{attribute 'qualified_only'}
VAR_GLOBAL
	
	// Termo-resistances outputs
	O_TermL:BOOL;
	O_TermU:BOOL;
END_VAR

(* stored: Version 1.1.0.1, ProductVersion 3.1.4024.9
   GVL IO: Id {f19c6e7d-dfbd-4478-b507-c13927482bf7} *)
